PROGRAM JSON_decode
VAR
	mydata : sensorData;
	fixedMessage : STRING(150) := '{"id": "4CCE8E","battery": 80,"flag": 0,"mode": 1,"temp": 23,"hum": 0}';
	//block
	fbJson		: FB_JsonDomParser;
	//parsed
	parsedDoc	: SJsonValue;
	parsedVal	: SJsonValue;

END_VAR

// rx
parsedDoc := fbJson.ParseDocument(fixedMessage);

parsedVal := fbJson.FindMember(parsedDoc, 'id');
mydata.id := fbJson.GetString(parsedVal);

parsedVal := fbJson.FindMember(parsedDoc, 'battery');
mydata.battery := fbJson.GetInt(parsedVal);

parsedVal := fbJson.FindMember(parsedDoc, 'flag');
mydata.flag := fbJson.GetInt(parsedVal);

parsedVal := fbJson.FindMember(parsedDoc, 'mode');
mydata.mode := fbJson.GetInt(parsedVal);

parsedVal := fbJson.FindMember(parsedDoc, 'temp');
mydata.temp := fbJson.GetInt(parsedVal);

parsedVal := fbJson.FindMember(parsedDoc, 'hum');
mydata.hum := fbJson.GetInt(parsedVal);
(*
parsedVal2 := fbJson.FindMember(parsedVal1, 'battery');
mydata.battery := fbJson.GetString(parsedVal);

parsedVal3 := fbJson.FindMember(parsedVal2, 'flag');
mydata.flag := fbJson.GetString(parsedVal);

parsedVal4 := fbJson.FindMember(parsedVal3, 'mode');
mydata.mode := fbJson.GetString(parsedVal);

parsedVal5 := fbJson.FindMember(parsedVal4, 'temp');
mydata.temp := fbJson.GetString(parsedVal);

parsedVal6 := fbJson.FindMember(parsedVal5, 'hum');
mydata.hum := fbJson.GetString(parsedVal);*)

END_PROGRAM

(* stored: Version 1.1.0.1, ProductVersion 3.1.4024.0
   POU JSON_decode: Id {8e01a1e0-72a7-4677-b34c-52a05cbdaae2}, SpecialFunc None *)
